INTERFACE I_VisitibleElement

METHOD accept
VAR_INPUT
	in_ipVisitor	: I_Visitor;
END_VAR
END_METHOD

END_INTERFACE

(* stored: Version 1.1.0.1
   Itf I_VisitibleElement: Id {07de59f1-ba5f-4884-8b50-b7eaabf92cec}
   Method accept: Id {23533864-0678-4ece-bfb5-467e70d72165} *)
